// TIA Portal V20 export
// export: Created 2025-12-01T14:57:08.432378Z, ExportSetting None, DisplayName Totally Integrated Automation Portal, DisplayVersion V20 Update 3, DisplayName TIA Portal Openness, DisplayVersion V20 Update 3, DisplayName TIA Portal Version Control Interface, DisplayVersion V20 Update 3, DisplayName STEP 7 Professional, DisplayVersion V20 Update 3, DisplayName STEP 7 Safety, DisplayVersion V20 Update 2, DisplayName WinCC Basic/Comfort/Advanced, DisplayVersion V20 Update 3, DisplayName WinCC Professional, DisplayVersion V20 Update 3, DisplayName WinCC Unified, DisplayVersion V20 Update 3
FUNCTION "FC826_CalcularOrdenUT_MesaCruce" : Void   // FC826, STL
{ S7_Optimized_Access := 'FALSE' }
// stored: AutoNumber false
   VAR_INPUT
      NumeroUT : UInt;
   END_VAR
   VAR_OUTPUT
      Orden : Word;   // Orden a realizar en la MESA
      Auxiliar_01 : UInt;   // Auxiliar 01 de la Orden a realizar en la MESA
      MesaSalidaMulti : UInt;   // Auxiliar 02 de la Orden a realizar en la MESA
      Auxiliar_03 : UInt;   // Auxiliar 03 de la Orden a realizar en la MESA
      Auxiliar_04 : UInt;   // Auxiliar 04 de la Orden a realizar en la MESA
   END_VAR
   VAR_TEMP
      IndiceRutaUT : UInt;
      P_Temporal : DWord;
      MesaIntermedia : UInt;
      MesaRutaParcial : UInt;
      OrdenSalida : UInt;
      NumeroMesa : UInt;
      SiguienteUT : UInt;
      MesaEspera : UInt;
      OrdenTMP : Word;
      SinUT_EnMesa : Bool;
      RutaOK_EnMesa : Bool;
   END_VAR
BEGIN

NETWORK
TITLE = Inicializar
/////////////////////////////////////////////////////////////////////////
// Inicializaciones de las variables de los DB's

      L     0;
      T     #Orden;
      T     #OrdenTMP;
      T     #MesaSalidaMulti;
      T     #Auxiliar_01;
      T     #Auxiliar_03;
      T     #Auxiliar_04;


/////////////////////////////////////////////////////////////////////////
// Mesa Actual dentro del PLC
      L     "DB812_UTs_Control".UT[#NumeroUT].MesaActual;
      L     "CTE_OffsetMesa";
      -I;
      T     #NumeroMesa;



NETWORK
TITLE = Calcular Orden - FASE 01 >>> Ruta Para Continuar >>> Modificacion (07/05/2020)
/////////////////////////////////////////////////////////////////////////
// --- Es una Mesa de Cruce
/////////////////////////////////////////////////////////////////////////
// La mesa siguiente definida en la Mesa Actual, es una de salidas posibles
// Pero una vez encontrada la salida, debe cumplir unas condiciones:
// - Para enviar orden hay que ver si tiene que ESPERAR a que este LIBRE la
//   mesa SIGUIENTE (Mesa_Sxx) dependiendo de la salida definida
//   * Si tiene que esperar, no hacer nada
//   * Si no tiene que esperar, enviar orden y darla por tratada
//
// MODIFICACION (07/05/2020) --> Verificar si todas tienen RUTA
//
// MODIFICACION (06/05/2013) --> Nueva operativa   (ALON)
// - Buscar la mesa de salida de la ruta partiendo desde la ultima posición
//   utilizada.
//   Si no se encuentra, en esta parte de la ruta.
//   Se utilizara la ruta completa (Antigua operativa)
// OPERATIVA ANTIGUA
// - Recorrer toda la ruta, desde el principio buscando la mesa de salida
//
// - Si se envia la orden NO hay que quitar esta mesa de la ruta
//   Ya ha sido utilizada    (CAMBIO ALON - 24/10/2012)
/////////////////////////////////////////////////////////////////////////


/////////////////////////////////////////////////////////////////////////
/////////////////////////////////////////////////////////////////////////
/////////////////////////////////////////////////////////////////////////
// --- FASE 01, Mirar las rutas de las UT's de la Mesa
//     MODIFICACION AÑADIDO (07/05/2020)
      SET;
      A     "DB850_DefinicionMesas".Mesa[#NumeroMesa].ConfigMesa.RutaSalidaTodas;
      O     "DB850_DefinicionMesas".Mesa[#NumeroMesa].ConfigMesa.MultiplesCargasDeSalida;
      O     "DB850_DefinicionMesas".Mesa[#NumeroMesa].ConfigMesa.GrupoDeSalida;
      JCN   FinalControlRutaEnMesa;

// Esta parte cuidado recircular porque tiene el mismo destino
// Anulo por Ahora 2020 05 22
//      SET                        // Si tiene que recicular
//      U     #DatosUT.RecircularCarga
//      SPB   FinalControlRutaEnMesa

      CALL  "FC872_VerificarRutaEnMesa"
      ( Mesa      := #NumeroMesa,
        TestGrupo := "DB850_DefinicionMesas".Mesa[#NumeroMesa].ConfigMesa.GrupoDeSalida,
        RutaOK    := #RutaOK_EnMesa
      );

      SET;  // No tienen todas Ruta ?
      AN    #RutaOK_EnMesa;
      JC    FinalCalcularOrden;

/////////////////////////////////////////////////////////////////////////
// Tiene Ruta para Continuar - Final de FASE 02
FinalControlRutaEnMesa:NOP   0;



NETWORK
TITLE = Calcular Orden - FASE 02 >>> NUEVA OPERATIVA - Buscar por RUTA PARCIAL
/////////////////////////////////////////////////////////////////////////
/////////////////////////////////////////////////////////////////////////
/////////////////////////////////////////////////////////////////////////
// --- FASE 02, NUEVA OPERATIVA - Buscar por RUTA PARCIAL
//     MODIFICACION AÑADIDO (06/05/2013) RECIRCULACION
//     Buscar en que parte de la ruta se esta --> RUTA PARCIAL
//
//    Si no se encuentra >>> Se utilizara la Ruta Completa
//    Si se encuentra    >>> Se utilizara la Ruta Parcial


/////////////////////////////////////////////////////////////////////////
// 1. >>> Ultima Mesa tratada de la Ruta
      L     "DB812_UTs_Control".UT[#NumeroUT].MesaIntermedia;
      T     #MesaRutaParcial;


/////////////////////////////////////////////////////////////////////////
// 2. >>> Preparacion de la Ruta de la UT
      L     0;
      T     #IndiceRutaUT;


/////////////////////////////////////////////////////////////////////////
// 3. >>> Recorrer la Ruta haber si se encuentra donde se dejo
InicioBucleBusquedaInicial_EnRutaParcial:NOP   0;
      L     "DB813_UTs_Ruta".UT[#NumeroUT].Ruta[#IndiceRutaUT];
      T     #MesaIntermedia;  // Poner la nueva ruta intermedia

      L     #MesaIntermedia;  // No hay Mesa Intermedia ?
      L     0;
      ==I;  // No encontrado nada en la NUEVA OPERATIVA
      JC    FinalBucleBusqueda_EnRutaParcial;

      L     #MesaIntermedia;  // Mesa Intermedia = Mesa Ruta Parcial
      L     #MesaRutaParcial;
      ==I;  // Encontrado donde se dejo ACTIVAR NUEVA OPERATIVA
      JC    EnContradaMesa_EnRutaParcial;

      L     #MesaIntermedia;  // Se comprueba si es el Final de la Ruta
      L     "DB812_UTs_Control".UT[#NumeroUT].MesaDestino;
      ==I;  // No encontrado nada en la NUEVA OPERATIVA
      JC    FinalBucleBusqueda_EnRutaParcial;

// 3.F >>> Mesa Siguiente de la Ruta
      L     #IndiceRutaUT;
      L     1;
      +I;
      T     #IndiceRutaUT;
      JU    InicioBucleBusquedaInicial_EnRutaParcial;


/////////////////////////////////////////////////////////////////////////
// Encontrada Mesa Intermedia en RUTA PARCIAL
// NUEVA OPERATIVA (06/05/2013) RECIRCULACION
// Comprobar todas las Mesa de la Ruta PARCIAL, si esta definida alguna en la Mesa
EnContradaMesa_EnRutaParcial:NOP   0;


/////////////////////////////////////////////////////////////////////////
// 1. >>> Recorrer la Ruta haber si se encuentra, alguna Salida Definida
InicioBucleBusquedaFinal_EnRutaParcial:NOP   0;
      L     "DB813_UTs_Ruta".UT[#NumeroUT].Ruta[#IndiceRutaUT];
      T     #MesaIntermedia;  // Poner la nueva ruta intermedia

      L     #MesaIntermedia;  // No hay Mesa Intermedia ?
      L     0;
      ==I;  // No encontrado nada en la NUEVA OPERATIVA
      JC    FinalBucleBusqueda_EnRutaParcial;


/////////////////////////////////////////////////////////////////////////
// 2. >>> Comprobar cual es la mesa siguiente
//        Mesa_S01 = MesaIntermedia -> Salida por S1
//        Con Offset en la Condiguracion 28/03/2022
      L     1;  // Inicializo que sale
      T     #OrdenSalida;

      L     "DB850_DefinicionMesas".Mesa[#NumeroMesa].Mesa_S01;
//      L     "CTE_OffsetMesa"     // Mesa Correcta ?
//      +I                         // + Offset
      L     #MesaIntermedia;
      <>I;  // No es esta salida del Cruce
      JC    FinControlMesaSalida_S01_EnRutaParcial;

// --- Es esta salida del Cruce
// --- Comprobar si una Mesa de ESPERA
      SET;  // No es Salida de ESPERA ?
      AN    "DB850_DefinicionMesas".Mesa[#NumeroMesa].ConfigMesa.Espera_S01;
      JC    EnContradaMesaSalida_EnLaRuta;

// --- Mirar si Mesa_S01 esta Vacia
      L     "DB850_DefinicionMesas".Mesa[#NumeroMesa].Mesa_S01;
      L     "CTE_OffsetMesa";
      -I;  // --- Calculo de la Mesa en Espera 28/03/2022
      T     #MesaEspera;

      CALL  "FC870_MesaSinUT"
      ( Mesa  := #MesaEspera,
        SinUT := #SinUT_EnMesa
      );

      SET;  // Y la Mesa esta con UT ?
      AN    #SinUT_EnMesa;
      JC    FinalCalcularOrden;  // NO esta Vacia
      JU    EnContradaMesaSalida_EnLaRuta;

// --- Se acabo con la Mesa_S01
FinControlMesaSalida_S01_EnRutaParcial:NOP   0;


/////////////////////////////////////////////////////////////////////////
// 3. >>> Comprobar cual es la mesa siguiente
//        Mesa_S02 = MesaIntermedia -> Salida por S2
//        Con Offset en la Condiguracion 28/03/2022
      L     2;  // Inicializo que sale
      T     #OrdenSalida;

      L     "DB850_DefinicionMesas".Mesa[#NumeroMesa].Mesa_S02;
//      L     "CTE_OffsetMesa"     // Mesa Correcta ?
//      +I                         // + Offset
      L     #MesaIntermedia;
      <>I;  // No es esta salida del Cruce
      JC    FinControlMesaSalida_S02_EnRutaParcial;

// --- Es esta salida del Cruce
// --- Comprobar si una Mesa de ESPERA
      SET;  // No es Salida de ESPERA ?
      AN    "DB850_DefinicionMesas".Mesa[#NumeroMesa].ConfigMesa.Espera_S02;
      JC    EnContradaMesaSalida_EnLaRuta;

// --- Mirar si Mesa_S02 esta Vacia
      L     "DB850_DefinicionMesas".Mesa[#NumeroMesa].Mesa_S02;
      L     "CTE_OffsetMesa";
      -I;  // --- Calculo de la Mesa en Espera 28/03/2022
      T     #MesaEspera;

      CALL  "FC870_MesaSinUT"
      ( Mesa  := #MesaEspera,
        SinUT := #SinUT_EnMesa
      );

      SET;  // Y la Mesa esta con UT ?
      AN    #SinUT_EnMesa;
      JC    FinalCalcularOrden;  // NO esta Vacia
      JU    EnContradaMesaSalida_EnLaRuta;

// --- Se acabo con la Mesa_S02
FinControlMesaSalida_S02_EnRutaParcial:NOP   0;


/////////////////////////////////////////////////////////////////////////
// 4. >>> Comprobar cual es la mesa siguiente
//        Mesa_S03 = MesaIntermedia -> Salida por S3
//        Con Offset en la Condiguracion 28/03/2022
      L     3;  // Inicializo que sale por S3
      T     #OrdenSalida;

      L     "DB850_DefinicionMesas".Mesa[#NumeroMesa].Mesa_S03;
//      L     "CTE_OffsetMesa"     // Mesa Correcta ?
//      +I                         // + Offset
      L     #MesaIntermedia;
      <>I;  // No es esta salida del Cruce
      JC    FinControlMesaSalida_S03_EnRutaParcial;

// --- Es esta salida del Cruce
// --- Comprobar si una Mesa de ESPERA
      SET;  // No es Salida de ESPERA ?
      AN    "DB850_DefinicionMesas".Mesa[#NumeroMesa].ConfigMesa.Espera_S03;
      JC    EnContradaMesaSalida_EnLaRuta;

// --- Mirar si Mesa_S03 esta Vacia
      L     "DB850_DefinicionMesas".Mesa[#NumeroMesa].Mesa_S03;
      L     "CTE_OffsetMesa";
      -I;  // --- Calculo de la Mesa en Espera 28/03/2022
      T     #MesaEspera;

      CALL  "FC870_MesaSinUT"
      ( Mesa  := #MesaEspera,
        SinUT := #SinUT_EnMesa
      );

      SET;  // Y la Mesa esta con UT ?
      AN    #SinUT_EnMesa;
      JC    FinalCalcularOrden;  // NO esta Vacia
      JU    EnContradaMesaSalida_EnLaRuta;

// --- Se acabo con la Mesa_S03
FinControlMesaSalida_S03_EnRutaParcial:NOP   0;


/////////////////////////////////////////////////////////////////////////
// 5. >>> Comprobar cual es la mesa siguiente
//        Mesa_S04 = MesaIntermedia -> Salida por S4
//        Con Offset en la Condiguracion 28/03/2022
      L     4;  // Inicializo que sale
      T     #OrdenSalida;

      L     "DB850_DefinicionMesas".Mesa[#NumeroMesa].Mesa_S04;
//      L     "CTE_OffsetMesa"     // Mesa Correcta ?
//      +I                         // + Offset
      L     #MesaIntermedia;
      <>I;  // No es esta salida del Cruce
      JC    FinControlMesaSalida_S04_EnRutaParcial;

// --- Es esta salida del Cruce
// --- Comprobar si una Mesa de ESPERA
      SET;  // No es Salida de ESPERA ?
      AN    "DB850_DefinicionMesas".Mesa[#NumeroMesa].ConfigMesa.Espera_S04;
      JC    EnContradaMesaSalida_EnLaRuta;

// --- Mirar si Mesa_S04 esta Vacia
      L     "DB850_DefinicionMesas".Mesa[#NumeroMesa].Mesa_S04;
      L     "CTE_OffsetMesa";
      -I;  // --- Calculo de la Mesa en Espera 28/03/2022
      T     #MesaEspera;

      CALL  "FC870_MesaSinUT"
      ( Mesa  := #MesaEspera,
        SinUT := #SinUT_EnMesa
      );

      SET;  // Y la Mesa esta con UT ?
      AN    #SinUT_EnMesa;
      JC    FinalCalcularOrden;  // NO esta Vacia
      JU    EnContradaMesaSalida_EnLaRuta;

// --- Se acabo con la Mesa_S04
FinControlMesaSalida_S04_EnRutaParcial:NOP   0;


/////////////////////////////////////////////////////////////////////////
// 6. >>> Seguir recorriendo la RUTA PARCIAL

      L     #MesaIntermedia;  // Se comprueba si es el Final de la Ruta
      L     "DB812_UTs_Control".UT[#NumeroUT].MesaDestino;
      ==I;  // No encontrado nada en la NUEVA OPERATIVA
      JC    FinalBucleBusqueda_EnRutaParcial;

// --- Mesa Siguiente de la Ruta
      L     #IndiceRutaUT;
      L     1;
      +I;
      T     #IndiceRutaUT;
      JU    InicioBucleBusquedaFinal_EnRutaParcial;


/////////////////////////////////////////////////////////////////////////
/////////////////////////////////////////////////////////////////////////
/////////////////////////////////////////////////////////////////////////


/////////////////////////////////////////////////////////////////////////
/////////////////////////////////////////////////////////////////////////
/////////////////////////////////////////////////////////////////////////
// Final de la FASE 02 : No Encontrada >>> Utilizar RUTA COMPLETA
// RUTA PARCIAL INSUFICIENTE --> Mirar RUTA TOTAL
FinalBucleBusqueda_EnRutaParcial:NOP   0;



NETWORK
TITLE = Calcular Orden - FASE 03 >>> ANTIGUA OPERATIVA - Buscar por RUTA COMPLETA
/////////////////////////////////////////////////////////////////////////
/////////////////////////////////////////////////////////////////////////
/////////////////////////////////////////////////////////////////////////
// --- FASE 03, ANTIGUA OPERATIVA - Buscar por RUTA COMPLETA
// --- Comprobobar todas las Mesas de la Ruta,
//     si esta definida alguna en la mesa
// --- OPERATIVA (24/10/2012)


/////////////////////////////////////////////////////////////////////////
// 1. >>> Preparacion de la Ruta de la UT
      L     0;
      T     #IndiceRutaUT;


/////////////////////////////////////////////////////////////////////////
// 2. >>> Recorrer la Ruta haber si se encuentra, alguna Salida Definida
InicioBucleBusqueda_EnRutaCompleta:NOP   0;
      L     "DB813_UTs_Ruta".UT[#NumeroUT].Ruta[#IndiceRutaUT];
      T     #MesaIntermedia;  // Poner la nueva ruta intermedia

      L     #MesaIntermedia;  // No hay Mesa Intermedia ?
      L     0;
      ==I;  // No esta en Ruta, Pedir Ruta
      JC    PedirRutaNueva_FueraDeRuta;


/////////////////////////////////////////////////////////////////////////
// 3. >>> Comprobar cual es la mesa siguiente
//        Mesa_S01 = MesaIntermedia -> Salida por S1
//        Con Offset en la Condiguracion 28/03/2022
      L     1;  // Inicializo que sale
      T     #OrdenSalida;

      L     "DB850_DefinicionMesas".Mesa[#NumeroMesa].Mesa_S01;
//      L     "CTE_OffsetMesa"     // Mesa Correcta ?
//      +I                         // + Offset
      L     #MesaIntermedia;
      <>I;  // No es esta salida del Cruce
      JC    FinControlMesaSalida_S01_EnRutaCompleta;

// --- Es esta salida del Cruce
// --- Comprobar si una Mesa de ESPERA
      SET;  // No es Salida de ESPERA ?
      AN    "DB850_DefinicionMesas".Mesa[#NumeroMesa].ConfigMesa.Espera_S01;
      JC    EnContradaMesaSalida_EnLaRuta;

// --- Mirar si Mesa_S01 esta Vacia
      L     "DB850_DefinicionMesas".Mesa[#NumeroMesa].Mesa_S01;
      L     "CTE_OffsetMesa";
      -I;  // --- Calculo de la Mesa en Espera 28/03/2022
      T     #MesaEspera;

      CALL  "FC870_MesaSinUT"
      ( Mesa  := #MesaEspera,
        SinUT := #SinUT_EnMesa
      );

      SET;  // Y la Mesa esta con UT ?
      AN    #SinUT_EnMesa;
      JC    FinalCalcularOrden;  // NO esta Vacia
      JU    EnContradaMesaSalida_EnLaRuta;

// --- Se acabo con la Mesa_S01
FinControlMesaSalida_S01_EnRutaCompleta:NOP   0;


/////////////////////////////////////////////////////////////////////////
// 4. >>> Comprobar cual es la mesa siguiente
//        Mesa_S02 = MesaIntermedia -> Salida por S2
//        Con Offset en la Condiguracion 28/03/2022
      L     2;  // Inicializo que sale
      T     #OrdenSalida;

      L     "DB850_DefinicionMesas".Mesa[#NumeroMesa].Mesa_S02;
//      L     "CTE_OffsetMesa"     // Mesa Correcta ?
//      +I                         // + Offset
      L     #MesaIntermedia;
      <>I;  // No es esta salida del Cruce
      JC    FinControlMesaSalida_S02_EnRutaCompleta;

// --- Es esta salida del Cruce
// --- Comprobar si una Mesa de ESPERA
      SET;  // No es Salida de ESPERA ?
      AN    "DB850_DefinicionMesas".Mesa[#NumeroMesa].ConfigMesa.Espera_S02;
      JC    EnContradaMesaSalida_EnLaRuta;

// --- Mirar si Mesa_S02 esta Vacia
      L     "DB850_DefinicionMesas".Mesa[#NumeroMesa].Mesa_S02;
      L     "CTE_OffsetMesa";
      -I;  // --- Calculo de la Mesa en Espera 28/03/2022
      T     #MesaEspera;

      CALL  "FC870_MesaSinUT"
      ( Mesa  := #MesaEspera,
        SinUT := #SinUT_EnMesa
      );

      SET;  // Y la Mesa esta con UT ?
      AN    #SinUT_EnMesa;
      JC    FinalCalcularOrden;  // NO esta Vacia
      JU    EnContradaMesaSalida_EnLaRuta;

// --- Se acabo con la Mesa_S02
FinControlMesaSalida_S02_EnRutaCompleta:NOP   0;


/////////////////////////////////////////////////////////////////////////
// 5. >>> Comprobar cual es la mesa siguiente
//        Mesa_S03 = MesaIntermedia -> Salida por S3
//        Con Offset en la Condiguracion 28/03/2022
      L     3;  // Inicializo que sale por S3
      T     #OrdenSalida;

      L     "DB850_DefinicionMesas".Mesa[#NumeroMesa].Mesa_S03;
//      L     "CTE_OffsetMesa"     // Mesa Correcta ?
//      +I                         // + Offset
      L     #MesaIntermedia;
      <>I;  // No es esta salida del Cruce
      JC    FinControlMesaSalida_S03_EnRutaCompleta;

// --- Es esta salida del Cruce
// --- Comprobar si una Mesa de ESPERA
      SET;  // No es Salida de ESPERA ?
      AN    "DB850_DefinicionMesas".Mesa[#NumeroMesa].ConfigMesa.Espera_S03;
      JC    EnContradaMesaSalida_EnLaRuta;

// --- Mirar si Mesa_S03 esta Vacia
      L     "DB850_DefinicionMesas".Mesa[#NumeroMesa].Mesa_S03;
      L     "CTE_OffsetMesa";
      -I;  // --- Calculo de la Mesa en Espera 28/03/2022
      T     #MesaEspera;

      CALL  "FC870_MesaSinUT"
      ( Mesa  := #MesaEspera,
        SinUT := #SinUT_EnMesa
      );

      SET;  // Y la Mesa esta con UT ?
      AN    #SinUT_EnMesa;
      JC    FinalCalcularOrden;  // NO esta Vacia
      JU    EnContradaMesaSalida_EnLaRuta;

// --- Se acabo con la Mesa_S03
FinControlMesaSalida_S03_EnRutaCompleta:NOP   0;


/////////////////////////////////////////////////////////////////////////
// 6. >>> Comprobar cual es la mesa siguiente
//        Mesa_S04 = MesaIntermedia -> Salida por S4
//        Con Offset en la Condiguracion 28/03/2022
      L     4;  // Inicializo que sale
      T     #OrdenSalida;

      L     "DB850_DefinicionMesas".Mesa[#NumeroMesa].Mesa_S04;
//      L     "CTE_OffsetMesa"     // Mesa Correcta ?
//      +I                         // + Offset
      L     #MesaIntermedia;
      <>I;  // No es esta salida del Cruce
      JC    FinControlMesaSalida_S04_EnRutaCompleta;

// --- Es esta salida del Cruce
// --- Comprobar si una Mesa de ESPERA
      SET;  // No es Salida de ESPERA ?
      AN    "DB850_DefinicionMesas".Mesa[#NumeroMesa].ConfigMesa.Espera_S04;
      JC    EnContradaMesaSalida_EnLaRuta;

// --- Mirar si Mesa_S04 esta Vacia
      L     "DB850_DefinicionMesas".Mesa[#NumeroMesa].Mesa_S04;
      L     "CTE_OffsetMesa";
      -I;  // --- Calculo de la Mesa en Espera 28/03/2022
      T     #MesaEspera;

      CALL  "FC870_MesaSinUT"
      ( Mesa  := #MesaEspera,
        SinUT := #SinUT_EnMesa
      );

      SET;  // Y la Mesa esta con UT ?
      AN    #SinUT_EnMesa;
      JC    FinalCalcularOrden;  // NO esta Vacia
      JU    EnContradaMesaSalida_EnLaRuta;

// --- Se acabo con la Mesa_S04
FinControlMesaSalida_S04_EnRutaCompleta:NOP   0;


/////////////////////////////////////////////////////////////////////////
// 7. >>> Seguir recorriendo la RUTA Completa

      L     #MesaIntermedia;  // Se comprueba si es el Final de la Ruta
      L     "DB812_UTs_Control".UT[#NumeroUT].MesaDestino;
      ==I;  // No encontrado nada en la NUEVA OPERATIVA
      JC    PedirRutaNueva_FueraDeRuta;

// --- Mesa Siguiente de la Ruta
      L     #IndiceRutaUT;
      L     1;
      +I;
      T     #IndiceRutaUT;
      JU    InicioBucleBusqueda_EnRutaCompleta;


/////////////////////////////////////////////////////////////////////////
/////////////////////////////////////////////////////////////////////////
/////////////////////////////////////////////////////////////////////////


/////////////////////////////////////////////////////////////////////////
/////////////////////////////////////////////////////////////////////////
/////////////////////////////////////////////////////////////////////////
// Final de la FASE 03 : Encontrada Mesa de Salida
FinalBucleBusqueda_EnRutaCompleta:NOP   0;
      JU    EnContradaMesaSalida_EnLaRuta;



NETWORK
TITLE = Calcular Orden - FASE 04 >>> Encontrada Mesa de Salida En la Ruta
/////////////////////////////////////////////////////////////////////////
/////////////////////////////////////////////////////////////////////////
/////////////////////////////////////////////////////////////////////////
// --- FASE 04, Encontrada Mesa de Salida En la Ruta
// --- Primero, doy por tratada la causa
// --- Segundo, Activarse la Mesa de Salida que Corresponda "OrdenSalida"
EnContradaMesaSalida_EnLaRuta:NOP   0;


/////////////////////////////////////////////////////////////////////////
// 1 >>> Doy por tratada la Mesa la Primera de la Mesa
      L     0;  // Dar por tratada
      T     "DB812_UTs_Control".UT[#NumeroUT].EstadoRecepcionUT;
      T     "DB812_UTs_Control".UT[#NumeroUT].EstadoEventoRecibido;

      L     #MesaIntermedia;
      T     "DB812_UTs_Control".UT[#NumeroUT].MesaIntermedia;

      SET;  // Reset - Recircular la Carga - Memoria del Retirar
      R     "DB812_UTs_Control".UT[#NumeroUT].AtributosDeLaUT.RecircularCarga;


/////////////////////////////////////////////////////////////////////////
// 2 >>> Si hay que darla por tratadas todas las de la Mesa

      SET;  // Hay que Recorrer el Resto de UTs de la Mesa
      AN    "DB850_DefinicionMesas".Mesa[#NumeroMesa].ConfigMesa.MultiplesCargasDeSalida;
      AN    "DB850_DefinicionMesas".Mesa[#NumeroMesa].ConfigMesa.GrupoDeSalida;
      JC    FinalBucleUTs_EnMesa;

      L     "DB812_UTs_Control".UT[#NumeroUT].UT_SiguienteMesa;
      T     #SiguienteUT;


InicioBucleUTs_EnMesa:NOP   0;
      L     #SiguienteUT;
      L     0;
      ==I;  // Hay mas UT's
      JC    FinalBucleUTs_EnMesa;

// Testear Grupo ?
      SET;
      AN    "DB850_DefinicionMesas".Mesa[#NumeroMesa].ConfigMesa.GrupoDeSalida;
      JC    ContinuarBucleUTs_EnMesa;

// Dar por tratado solo lo del mismo Grupo
// Grupo Primera UT == Grupo de la Siguiente
      L     "DB812_UTs_Control".UT[#NumeroUT].Grupo;
      L     "DB812_UTs_Control".UT[#SiguienteUT].Grupo;
      <>I;
      JC    FinalBucleUTs_EnMesa;

// Dar por tratada la Siguinete UT
ContinuarBucleUTs_EnMesa:NOP   0;
      L     0;  // Dar por tratada
      T     "DB812_UTs_Control".UT[#SiguienteUT].EstadoRecepcionUT;
      T     "DB812_UTs_Control".UT[#SiguienteUT].EstadoEventoRecibido;

      L     #MesaIntermedia;
      T     "DB812_UTs_Control".UT[#SiguienteUT].MesaIntermedia;

      SET;  // Reset - Recircular la Carga - Memoria del Retirar
      R     "DB812_UTs_Control".UT[#NumeroUT].AtributosDeLaUT.RecircularCarga;

      L     "DB812_UTs_Control".UT[#SiguienteUT].UT_SiguienteMesa;
      T     #SiguienteUT;
      JU    InicioBucleUTs_EnMesa;


/////////////////////////////////////////////////////////////////////////
// 2. >>> Final del Bucle
FinalBucleUTs_EnMesa:NOP   0;


/////////////////////////////////////////////////////////////////////////
// 3. >>>   Activarse la Mesa de Salida que Corresponda
//          En variable "OrdenSalida"

      L     #OrdenSalida;
      JL    SinOrden_Defecto;

// 3.1. Distribucion de la Orden de Salida
      JU    SinOrden_Defecto;  // OrdenSalida = 0
      JU    OrdenSalida_S01;  // OrdenSalida = 1
      JU    OrdenSalida_S02;  // OrdenSalida = 2
      JU    OrdenSalida_S03;  // OrdenSalida = 3
      JU    OrdenSalida_S04;  // OrdenSalida = 4

// 3.2. >>>> CUIDADO si llega aqui MALO es IMPOSIBLE
SinOrden_Defecto:NOP   0;
      JU    FinalCalcularOrden;



NETWORK
TITLE = Control - No existe Mesa de Salida - FUERA de RUTA
/////////////////////////////////////////////////////////////////////////
// --- No existe Mesa de Salida posible
//     La UT esta FUERA de RUTA
//     Realiazar, Evento de Pedir Ruta

PedirRutaNueva_FueraDeRuta:NOP   0;
      L     "DB812_UTs_Control".UT[#NumeroUT].EstadoGeneralUT;
      L     0;
      <>I;  //NO esta LIBRE?
      JC    FinalCalcularOrden;

      L     26;  // 26 - Generar Evento Pedir Ruta (FUERA DE RUTA)
      T     "DB812_UTs_Control".UT[#NumeroUT].EstadoGeneralUT;
      L     0;  // Dar por tratada
      T     "DB812_UTs_Control".UT[#NumeroUT].EstadoRecepcionUT;

      JU    FinalCalcularOrden;



NETWORK
TITLE = Generar Orden de Salida
/////////////////////////////////////////////////////////////////////////
/////////////////////////////////////////////////////////////////////////
// --- Ordenes a enviar dependiendo por donde sale
// --- Salida por S01
OrdenSalida_S01:NOP   0;
      L     P##OrdenTMP;
      L     P#0.1;
      +D;
      T     #P_Temporal;

      SET;  // Orden -> Activar Bit 1
      S     L [#P_Temporal];
      JU    FinalOrdenSalida;


/////////////////////////////////////////////////////////////////////////
/////////////////////////////////////////////////////////////////////////
// --- Ordenes a enviar dependiendo por donde sale
// --- Salida por S02
OrdenSalida_S02:NOP   0;
      L     P##OrdenTMP;
      L     P#0.2;
      +D;
      T     #P_Temporal;

      SET;  // Orden -> Activar Bit 2
      S     L [#P_Temporal];
      JU    FinalOrdenSalida;


/////////////////////////////////////////////////////////////////////////
/////////////////////////////////////////////////////////////////////////
// --- Ordenes a enviar dependiendo por donde sale
// --- Salida por S03
OrdenSalida_S03:NOP   0;
      L     P##OrdenTMP;
      L     P#0.3;
      +D;
      T     #P_Temporal;

      SET;  // Orden -> Activar Bit 3
      S     L [#P_Temporal];
      JU    FinalOrdenSalida;


/////////////////////////////////////////////////////////////////////////
/////////////////////////////////////////////////////////////////////////
// --- Ordenes a enviar dependiendo por donde sale
// --- Salida por S04
OrdenSalida_S04:NOP   0;
      L     P##OrdenTMP;
      L     P#0.4;
      +D;
      T     #P_Temporal;

      SET;  // Orden -> Activar Bit 4
      S     L [#P_Temporal];
      JU    FinalOrdenSalida;



/////////////////////////////////////////////////////////////////////////
/////////////////////////////////////////////////////////////////////////
// --- Ordenes a enviar dependiendo por donde sale
// --- Salida por Defecto
OrdenSalida_Defecto:NOP   0;
      L     P##OrdenTMP;
      L     P#0.5;
      +D;
      T     #P_Temporal;

      SET;  // Orden -> Activar Bit 5
      S     L [#P_Temporal];
      JU    FinalOrdenSalida;


/////////////////////////////////////////////////////////////////////////
/////////////////////////////////////////////////////////////////////////
// No Existen mas posibilidades
FinalOrdenSalida:NOP   0;



NETWORK
TITLE = Final de Calcular Orden
/////////a////////////////////////////////////////////////////////////////
// Finalizar la Funcion
FinalCalcularOrden:NOP   0;

      L     #OrdenTMP;
      T     #Orden;


END_FUNCTION
